PROGRAM MAIN
VAR
END_VAR

END_PROGRAM

(* stored: Version 1.1.0.1
   POU MAIN: Id {6dd2527d-7fb2-444c-afaa-6b697e55f349} *)
